FUNCTION_BLOCK IVController EXTENDS TcoCore.TcoComponent
VAR
    _triggerSensorTask        : TriggerSensor(THIS^);
    _readTool1CoordinatesTask : ReadCoordinates(THIS^, CoeIndex := Tool1CoeIndex);
    _readTool2CoordinatesTask : ReadCoordinates(THIS^, CoeIndex := Tool2CoeIndex);
    _readTool3CoordinatesTask : ReadCoordinates(THIS^, CoeIndex := Tool3CoeIndex);
    _calculationTask          : CalculationTask
    (
        THIS^
        , ResolutionX := 1280
        , ResolutionY := 960
        , OffsetX     := -5.57888
        , GainX       := 3.387877
        , OffsetY     := -70129
        , GainY       := 2.5438
    );
END_VAR

VAR
    _fb_coe_write       : FB_EcCoESdoWrite; // Function Block for writing in CoE
    _fb_coe_read        : FB_EcCoESdoRead;  // Function Block for reading from CoE
    userNetId           : T_AmsNetId;       // Have to be entered
    _startWrite         : BOOL := FALSE;    // Sign for start writing
    _startRead          : BOOL := FALSE;    // Sign for start reading
    _nState             : BYTE := 0;        // RW-status
    _int16Buffer        : INT;              // Buffer for reading
    _uint16Buffer       : UINT := 22;       // Buffer for writing
    _bTxPDOState AT %I* : BOOL;             // (PDO for synchronization)
    AdsErrId            : UDINT;
    CANopenErrId        : UDINT;

    _index             : UINT := 16#1008;
    _subIndex          : BYTE := 0;
    _result            : STRING;
    _stringBuffer      : STRING;
    _numberBuffer      : UDINT;
    _exe               : BOOL;
    _generalDeviceInfo : GeneralDeviceInformation;
    _IdentityCoe       : IdentityCoe;
    _coordinates       : Coordinates;
    _readCoordinates   : BOOL;
END_VAR
VAR CONSTANT
    Tool1CoeIndex : UINT := 16#8015;
    Tool2CoeIndex : UINT := 16#8025;
    Tool3CoeIndex : UINT := 16#8035;

END_VAR
VAR

    //    //Ethercat Status
    //~
    StatusOfSystem AT %I* : Status_of_System;
    //PDO Vision Sensor   
    InputResponse                                 AT %I* : Input_Response;
    ID01_CurrentValue                             AT %I* : ID01_Current_Value;
    ID02_MatchingRateOfPositionAdujustmentTool_01 AT %I* : ID02_Current_Value; //value 0..1
    ID03_MatchingRateOfPositionAdujustmentTool_02 AT %I* : ID03_Current_Value; //value 0..1
    ID04_MatchingRateOfPositionAdujustmentTool_03 AT %I* : ID04_Current_Value; //value 0..1
    ID05_MatchingRateOfPositionAdujustmentTool_04 AT %I* : ID05_Current_Value; //value 0..1
    ID06_MatchingRateOfPositionAdujustmentTool_05 AT %I* : ID06_Current_Value; //value 0..1
    ID07_MatchingRateOfPositionAdujustmentTool_06 AT %I* : ID07_Current_Value; //value 0..1
    ID08_MatchingRateOfPositionAdujustmentTool_07 AT %I* : ID08_Current_Value; //value 0..1
    ID01Status                                    AT %I* : ID01_Status;
    ID02Status                                    AT %I* : ID02_Status;
    ID03Status                                    AT %I* : ID03_Status;
    ID04Status                                    AT %I* : ID04_Status;
    ID05Status                                    AT %I* : ID05_Status;
    ID06Status                                    AT %I* : ID06_Status;
    ID07Status                                    AT %I* : ID07_Status;
    ID08Status                                    AT %I* : ID08_Status;
    InputRequest                                  AT %Q* : Input_Request;
    //    //General Ethercat Data
    WcState  AT %I* : WcState_0B2B16F9;
    InfoData AT %I* : InfoData;
    //~

    _trigger        : BOOL;
    _readString     : BOOL;
    _readDeviceInfo : BOOL;
END_VAR

////////////////////////////////////////////
_triggerSensorTask
(
    Iv3InputRequest1    := THIS^.InputRequest.Request_1
    , Iv3InputResponse1 := THIS^.InputResponse.Response_1
    , StatusOfSystem    := THIS^.StatusOfSystem
    , ActionDesc        := '<#TriggerSensor#>'
);

_readTool1CoordinatesTask
(
    InfoData         := THIS^.InfoData
    , StatusOfSystem := THIS^.StatusOfSystem
    , ResultValue    := THIS^.ID02_MatchingRateOfPositionAdujustmentTool_01.Tool_00_Score
    , ActionDesc     := '<#ReadCoordinates Tool1#>'
);

_readTool2CoordinatesTask
(
    InfoData         := THIS^.InfoData
    , StatusOfSystem := THIS^.StatusOfSystem
    , ResultValue    := THIS^.ID03_MatchingRateOfPositionAdujustmentTool_02.Tool_01_Score
    , ActionDesc     := '<#ReadCoordinates Tool2#>'
);

_readTool3CoordinatesTask
(
    InfoData         := THIS^.InfoData
    , StatusOfSystem := THIS^.StatusOfSystem
    , ResultValue    := THIS^.ID04_MatchingRateOfPositionAdujustmentTool_03.Tool_02_Score
    , ActionDesc     := '<#ReadCoordinates Tool3#>'
);

_calculationTask
(
    InfoData           := THIS^.InfoData
    , StatusOfSystem   := THIS^.StatusOfSystem
    , CoordinatesTool1 := _readTool1CoordinatesTask.RawCoordinates
    , CoordinatesTool2 := _readTool2CoordinatesTask.RawCoordinates
    , CoordinatesTool3 := _readTool3CoordinatesTask.RawCoordinates
    , ActionDesc       := '<#_calculationTask#>'
);

/////////////////////////////////////////////
//IF _trigger THEN
//    THIS^.InputRequest.Request_1.Trigger := TRUE;

//    IF THIS^.InputResponse.Response_1.Trigger THEN
//        _trigger                             := FALSE;
//        THIS^.InputRequest.Request_1.Trigger := FALSE;
//    end_if
//END_IF

userNetId := Tc2_System.F_CreateAmsNetId(THIS^.InfoData.AdsAddr.netId);

IF _readString THEN
    _stringBuffer := CoeReadString(_index := _index, _subIndex := _subIndex);
END_IF

IF _readDeviceInfo THEN

    IF GeneralDeviceInfo() THEN
        _readDeviceInfo := false;
    END_IF
END_IF

CoeReadIdentity();

IF _readCoordinates THEN
    IF CoeReadCoordinates() THEN
        _readCoordinates := FALSE;
    END_IF

END_IF

METHOD CalculationMethod : TcoCore.ITcoTaskStatus
IF (CalculationTask <> 0) THEN
    CalculationMethod := CalculationTask.Invoke();
END_IF
END_METHOD

PROPERTY CalculationTask : TcoCore.ITcoTask
GET
CalculationTask := _calculationTask;
END_GET
END_PROPERTY

METHOD CoeReadCoordinates : BOOL
VAR_INST
    step : UINT := 1;

END_VAR
CASE step OF
    1:
        CoeReadCoordinates := FALSE;
        step               := 10;
    10:
        _coordinates.xValue := CoeReadUDINT
        (
            _index      := 16#8015
            , _subIndex := 16#11
        );

        IF NOT _fb_coe_read.bBusy THEN
            step := 20;
        END_IF
    20:
        _coordinates.yValue := CoeReadUDINT
        (
            _index      := 16#8015
            , _subIndex := 16#12
        );

        IF NOT _fb_coe_read.bBusy THEN
            step := 40;
        END_IF
    40:
        _coordinates.variableValue := CoeReadUDINT
        (
            _index      := 16#8015
            , _subIndex := 16#13
        );

        IF NOT _fb_coe_read.bBusy THEN
            step               := 1;
            CoeReadCoordinates := TRUE;
        END_IF
END_CASE
END_METHOD

METHOD CoeReadIdentity : UDINT
VAR_INST
    _fb_coe_read_ext   : Tc2_EtherCAT.FB_EcCoESdoReadEx;
    _timeout           : TIME := DEFAULT_ADS_TIMEOUT;
    _identityCoeToSwap : IdentityCoe;

    i     : UINT;
    _test : STRING;
END_VAR

// Read entry
_fb_coe_read_ext
(
    sNetId            := userNetId
    , nSlaveAddr      := InfoData.AdsAddr.port
    , nSubIndex       := 0
    , nIndex          := 16#1018
    , pDstBuf         := ADR(_identityCoeToSwap)
    , cbBufLen        := 32
    , bExecute        := true
    , tTimeout        := _timeout
    , bCompleteAccess := TRUE
);

IF _fb_coe_read.bError THEN
    _nState := 100; // Error case
ELSE

    IF NOT _fb_coe_read.bBusy THEN
        _IdentityCoe.ProductKey   := SHR(_identityCoeToSwap.ProductKey, 16);
        _IdentityCoe.VendorId     := SHR(_identityCoeToSwap.VendorId, 16);
        _IdentityCoe.Revision     := SHR(_identityCoeToSwap.Revision, 16);
        _IdentityCoe.SerialNumber := SHR(_identityCoeToSwap.SerialNumber, 16);
        _fb_coe_read(bExecute := FALSE);
        _readString := false;
    END_IF

END_IF
END_METHOD

METHOD CoeReadString : STRING
//VAR_INST
//    _stringBuffer : STRING;
//END_VAR
VAR_INPUT
    _index    : UINT;
    _subIndex : BYTE;
END_VAR

// Read entry
_fb_coe_read
(
    sNetId       := userNetId
    , nSlaveAddr := InfoData.AdsAddr.port
    //    , nSlaveAddr := 1001
    , nSubIndex := _subIndex
    , nIndex    := _index
    , pDstBuf   := ADR(_stringBuffer)
    , cbBufLen  := 12
    , bExecute  := true
    , tTimeout  := T#1S
);

IF _fb_coe_read.bError THEN
    AdsErrId := _fb_coe_read.nErrId;
ELSE
    IF NOT _fb_coe_read.bBusy THEN
        _fb_coe_read(bExecute := FALSE);
        _readString := false;
    END_IF
END_IF

CoeReadString := _stringBuffer;
END_METHOD

METHOD CoeReadUDINT : UDINT
//VAR_INST
//    _stringBuffer : STRING;
//END_VAR
VAR_INPUT
    _index    : UINT;
    _subIndex : BYTE;
END_VAR

// Read entry
_fb_coe_read
(
    sNetId       := userNetId
    , nSlaveAddr := InfoData.AdsAddr.port
    //    , nSlaveAddr := 1001
    , nSubIndex := _subIndex
    , nIndex    := _index
    , pDstBuf   := ADR(_numberBuffer)
    , cbBufLen  := 32
    , bExecute  := true
    , tTimeout  := T#1S
);

IF _fb_coe_read.bError THEN
    _nState := 100; // Error case
ELSE
    IF NOT _fb_coe_read.bBusy THEN
        _fb_coe_read(bExecute := FALSE);
        _readString := false;
    END_IF
END_IF

CoeReadUDINT := _numberBuffer;
END_METHOD

{attribute 'monitoring' := 'call'}
PROPERTY ErrorId : UINT
GET
ErrorId := THIS^.StatusOfSystem.Error_Code or _readTool1CoordinatesTask.ErrorId or _triggerSensorTask.ErrorId;
END_GET
END_PROPERTY

METHOD PRIVATE GeneralDeviceInfo : BOOL;
VAR_INST
    step : UINT := 1;

END_VAR
CASE step OF
    1:
        GeneralDeviceInfo := FALSE;
        step              := 10;
    10:
        _generalDeviceInfo.DeviceName := CoeReadString
        (
            _index      := 16#1008
            , _subIndex := 0
        );

        IF NOT _fb_coe_read.bBusy THEN
            step := 20;
        END_IF
    20:
        step := 25;
    25:
        _generalDeviceInfo.HardwareVersion := CoeReadString
        (
            _index      := 16#1009
            , _subIndex := 0
        );

        IF NOT _fb_coe_read.bBusy THEN
            step := 30;
        END_IF
    30:
        step := 35;
    35:
        _generalDeviceInfo.DeviceType := CoeReadUDINT
        (
            _index      := 16#1000
            , _subIndex := 0
        );

        IF NOT _fb_coe_read.bBusy THEN
            step := 40;
        END_IF
    40:
        GeneralDeviceInfo := FALSE;
        step              := 45;
    45:
        _generalDeviceInfo.SoftwareVersion := CoeReadString
        (
            _index      := 16#100A
            , _subIndex := 0
        );

        IF NOT _fb_coe_read.bBusy THEN
            step              := 1;
            GeneralDeviceInfo := TRUE;
        END_IF

END_CASE
END_METHOD

{attribute 'monitoring' := 'call'}
PROPERTY IsError : BOOL
GET
//collected Error from Tasks
IsError := statusOfSystem.Error_Status OR TriggerSensorTask.Error or ReadTool1CoordinatesTask.Error;
END_GET
END_PROPERTY

PROPERTY RawCoordinatesTool1 : REFERENCE TO Coordinates
GET
RawCoordinatesTool1 REF= _readTool1CoordinatesTask.RawCoordinates;
END_GET
END_PROPERTY

PROPERTY RawCoordinatesTool2 : REFERENCE TO Coordinates
GET
RawCoordinatesTool2 REF= _readTool2CoordinatesTask.RawCoordinates;
END_GET
END_PROPERTY

PROPERTY RawCoordinatesTool3 : REFERENCE TO Coordinates
GET
RawCoordinatesTool3 REF= _readTool3CoordinatesTask.RawCoordinates;
END_GET
END_PROPERTY

METHOD ReadTool1CoordinatesMethod : TcoCore.ITcoTaskStatus
IF (ReadTool1CoordinatesTask <> 0) THEN
    ReadTool1CoordinatesMethod := ReadTool1CoordinatesTask.Invoke();
END_IF
END_METHOD

PROPERTY ReadTool1CoordinatesTask : TcoCore.ITcoTask
GET
ReadTool1CoordinatesTask := _readTool1CoordinatesTask;
END_GET
END_PROPERTY

METHOD ReadTool2CoordinatesMethod : TcoCore.ITcoTaskStatus
IF (ReadTool2CoordinatesTask <> 0) THEN
    ReadTool2CoordinatesMethod := ReadTool2CoordinatesTask.Invoke();
END_IF
END_METHOD

PROPERTY ReadTool2CoordinatesTask : TcoCore.ITcoTask
GET
ReadTool2CoordinatesTask := _readTool2CoordinatesTask;
END_GET
END_PROPERTY

METHOD ReadTool3CoordinatesMethod : TcoCore.ITcoTaskStatus
IF (ReadTool3CoordinatesTask <> 0) THEN
    ReadTool3CoordinatesMethod := ReadTool3CoordinatesTask.Invoke();
END_IF
END_METHOD

PROPERTY ReadTool3CoordinatesTask : TcoCore.ITcoTask
GET
ReadTool3CoordinatesTask := _readTool3CoordinatesTask;
END_GET
END_PROPERTY

(*~
    <docu>
        <summary>
            Restore all tasks of this instance into initial state.
        </summary>
    </docu>
~*)
METHOD Restore : ITcoRestorable

IF (TriggerSensorTask <> 0) THEN
    TriggerSensorTask.Restore();
END_IF;

IF (ReadTool1CoordinatesTask <> 0) THEN
    ReadTool1CoordinatesTask.Restore();
END_IF;

//IF (WriteDataTask) <> 0 THEN
//    WriteDataTask.Restore();
//END_IF

//IF (LockTask) <> 0 THEN
//    LockTask.Restore();
//END_IF

//IF (ResetTask) <> 0 THEN
//    ResetTask.Restore();
//END_IF
END_METHOD

METHOD PROTECTED ServiceMode
END_METHOD

METHOD TriggerSensorMethod : TcoCore.ITcoTaskStatus
IF (TriggerSensorTask <> 0) THEN
    TriggerSensorMethod := TriggerSensorTask.Invoke();
END_IF
END_METHOD

PROPERTY TriggerSensorTask : TcoCore.ITcoTask
GET
TriggerSensorTask := _triggerSensorTask;
END_GET
END_PROPERTY

END_FUNCTION_BLOCK

(* stored: Version 1.1.0.1, ProductVersion 3.1.4024.12
   POU IVController: Id {dc97945e-e484-0055-193f-f0ad3a13ca29}, SpecialFunc None
   Folder old: Id {b26ebfb8-7b13-0ab2-293c-ccdc657e455d}
   Folder CoeActions: Id {38ad5833-e228-06d5-08c2-692a96a63a0e}
   Folder Operations: Id {73edbd5f-9d8c-0675-1377-2777718712ca}
   Folder Output: Id {49e001ad-6d3b-0279-17e3-1e208771d9e3}
   Folder Status: Id {88295d5c-9c9f-0625-38a0-8dbfe52d7dab}
   Folder Tasks: Id {d55a3cef-ea3c-0d2c-34c4-7b3b367731a4}
   Method CalculationMethod: Id {0c486270-ab06-0bd5-3aa6-e130a635c996}
   Property CalculationTask: Id {24e151f0-b3a5-0a0b-1f50-ff4b657074db}
   Get Get: Id {ad343cd0-a479-02bc-0b06-57d2460bd6fd}
   Method CoeReadCoordinates: Id {d69b9830-585e-0540-3a8c-20a136c13133}
   Method CoeReadIdentity: Id {e57c205c-7cb3-05a6-3726-236b1a9f2fa2}
   Method CoeReadString: Id {42f2292e-1927-0b19-3ef9-98e41834e163}
   Method CoeReadUDINT: Id {92682cd2-ba9e-0cfb-2606-7b5c3a5df8e8}
   Property ErrorId: Id {170082a8-5568-0cb7-25a9-5def9d9978a7}
   Get Get: Id {890deffe-5712-015b-2b21-50b154030c91}
   Method GeneralDeviceInfo: Id {537a1c31-cc9e-0538-0ff6-87339f8ab6f8}
   Property IsError: Id {fb44b890-472b-0194-0ca4-20bd3157b0fe}
   Get Get: Id {fc701666-5383-0ba7-10e6-e8194b7fc443}
   Property RawCoordinatesTool1: Id {0b90991a-a7c4-0005-17c3-92368e989ae1}
   Get Get: Id {800e7a61-3d57-0ef0-38e7-075359b444fa}
   Property RawCoordinatesTool2: Id {0e3a7a7b-f1dd-0d7f-3085-301da4e8e276}
   Get Get: Id {c32e2175-91b5-03c7-3c9d-a4668037ef39}
   Property RawCoordinatesTool3: Id {4e0c211f-e6ba-010e-1f01-3f24d4ab4dd6}
   Get Get: Id {5f3aa8fa-602f-0c4c-1e79-dcf4d263fdfa}
   Method ReadTool1CoordinatesMethod: Id {04f5c6d8-4ebf-00cf-269a-236b28b43364}
   Property ReadTool1CoordinatesTask: Id {872e3eb2-9d93-051b-005d-6c8a61bd7931}
   Get Get: Id {5ae01884-bf1c-0eb9-17fe-e61d84b630ef}
   Method ReadTool2CoordinatesMethod: Id {d908ec00-9575-09fd-2074-5207c89048ab}
   Property ReadTool2CoordinatesTask: Id {89ab5e87-1f52-0e78-014b-bec9c6ae13bf}
   Get Get: Id {48f65169-1fdd-0de1-373f-593e94f76835}
   Method ReadTool3CoordinatesMethod: Id {df71fc22-6c97-04d5-344f-cf11b5dd39a6}
   Property ReadTool3CoordinatesTask: Id {469512cc-7160-0114-27fc-d4485aa6830f}
   Get Get: Id {ed2f4a29-0e34-05aa-2354-89c64c99afe7}
   Method Restore: Id {427fb78b-85fe-0e6b-3852-1dca868a5299}
   Method ServiceMode: Id {f169ea65-2ad6-0a5f-2eee-aac69de0c435}
   Method TriggerSensorMethod: Id {791ded48-1e90-0e0d-2411-1b3167d67647}
   Property TriggerSensorTask: Id {cf021286-1fde-0b2d-24d9-ce6b04a60a41}
   Get Get: Id {a2d85624-9917-07dc-32d0-37b07774dd10} *)
